PROGRAM P3_06_CreateReport
VAR
	iStep					:INT;
	iError					:INT;
	tonResetError			:TON;
	trigStart				:R_TRIG;
	tonDelayStart			:TON;
	
	
	
	fbReport				:FB_PythonScript;
	fbSettingDelete			:FB_FileDelete;
	fbRecipeDelete			:FB_FileDelete;
	fbDeleteOldestBatch		:FB_DeleteOldestFile;
	fbSaveAsAlarm			:FB_FileSaveAs;
END_VAR


VAR PERSISTENT
	iReportsCreated			:INT;
END_VAR

ACT_CMDs();
tonResetError(IN:=(iError<>0),PT:=T#3S);
IF tonResetError.Q THEN
	iError:=0;
END_IF

trigStart(CLK:=GV.bBatchClose);

tonDelayStart(IN:=(iStep=10),PT:=T#1S);
CASE iStep OF
	
	0:
		IF trigStart.Q THEN
			iError:=0;
			iStep:=10;
		END_IF
		
	10:
		IF tonDelayStart.Q THEN
			iStep:=20;
		END_IF
		
	20:
		GV.stReport.bExport_Alarms:=TRUE;
		iStep:=25;
	25:
		IF NOT GV.stReport.bExport_Alarms THEN
			iStep:=30;
		END_IF
	26:
		GV.stReport.bSaveAs_Alarms:=TRUE;
		iStep:=27;
	27:
		IF NOT fbSaveAsAlarm.q_bBusy THEN
			iStep:=30;
		END_IF
		
	30:
		GV.stReport.bCreate_Report:=TRUE;
		IF fbReport.q_bBusy THEN
			iStep:=35;
		END_IF
	35:
		IF NOT fbReport.q_bBusy AND fbReport.q_bDone THEN
			iStep:=40;
		ELSIF fbReport.q_bError THEN
			iError:=iStep;
			iStep:=999;
		END_IF
	40:
		GV.stReport.bDelete_Data:=TRUE;
		iStep:=45;
	45:
		IF NOT GV.stReport.bDelete_Data THEN
			iStep:=50;
		END_IF
		
	50:
		GV.stReport.bDelete_OldestReport:=TRUE;
		IF fbDeleteOldestBatch.q_bBusy THEN
			iStep:=55;
		END_IF
	55:
		IF NOT fbDeleteOldestBatch.q_bBusy AND fbDeleteOldestBatch.q_bDone THEN
			iStep:=900;
		ELSIF fbDeleteOldestBatch.q_bError THEN
			iStep:=900;
			iError:=iStep;
		END_IF
		
	900:
		iReportsCreated:=iReportsCreated+1;
		GV.stReport.bStartSend_Sequence:=TRUE;
		iStep:=0;
	999:
		iStep:=0;
END_CASE

ACTION ACT_CMDs:
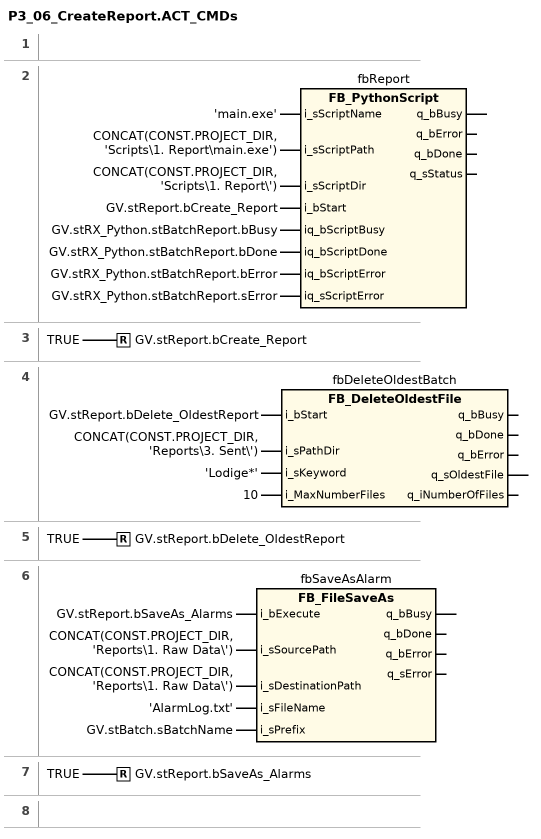
// NETWORK 1

// NETWORK 2
fbReport(
    i_sScriptName := 'main.exe',
    i_sScriptPath := CONCAT(CONST.PROJECT_DIR,'Scripts\1. Report\main.exe'),
    i_sScriptDir := CONCAT(CONST.PROJECT_DIR,'Scripts\1. Report\'),
    i_bStart := GV.stReport.bCreate_Report,
    iq_bScriptBusy := GV.stRX_Python.stBatchReport.bBusy,
    iq_bScriptDone := GV.stRX_Python.stBatchReport.bDone,
    iq_bScriptError := GV.stRX_Python.stBatchReport.bError,
    iq_sScriptError := GV.stRX_Python.stBatchReport.sError); // FB_PythonScript

// NETWORK 3
GV.stReport.bCreate_Report R= TRUE;

// NETWORK 4
fbDeleteOldestBatch(
    i_bStart := GV.stReport.bDelete_OldestReport,
    i_sPathDir := CONCAT(CONST.PROJECT_DIR,'Reports\3. Sent\'),
    i_sKeyword := 'Lodige*',
    i_MaxNumberFiles := 10); // FB_DeleteOldestFile

// NETWORK 5
GV.stReport.bDelete_OldestReport R= TRUE;

// NETWORK 6
fbSaveAsAlarm(
    i_bExecute := GV.stReport.bSaveAs_Alarms,
    i_sSourcePath := CONCAT(CONST.PROJECT_DIR,'Reports\1. Raw Data\'),
    i_sDestinationPath := CONCAT(CONST.PROJECT_DIR,'Reports\1. Raw Data\'),
    i_sFileName := 'AlarmLog.txt',
    i_sPrefix := GV.stBatch.sBatchName); // FB_FileSaveAs

// NETWORK 7
GV.stReport.bSaveAs_Alarms R= TRUE;

// NETWORK 8
END_ACTION

END_PROGRAM

(* stored: Version 1.1.0.1
   POU P3_06_CreateReport: Id {91230ed4-f090-42c4-80c1-92fe795f2356}, SpecialFunc None
   Action ACT_CMDs: Id {5be03143-2184-4a49-a951-3a18c79fe697} *)
